Staubli VAL3: remDisableArm.pgx

program remDisableArm(string& sReturn[] (dimensions=1))
begin
  // Turn the arm power OFF
  //
  logMsg("call remDisableArm")
  stopMove()
  resetMotion()
  disablePower()
  wait(isPowered()==false)
  sReturn="CMDDISABLEARM"
  logMsg("Arm power is DISABLED!")
end
